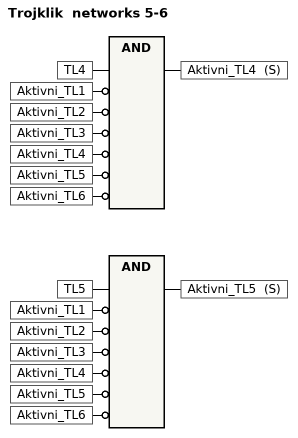
[picture p24: Trojklik (FBD) networks 5-6]
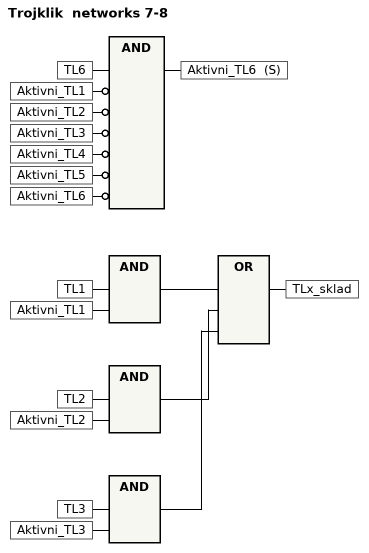
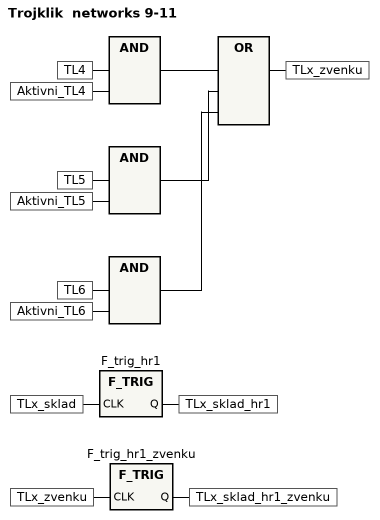
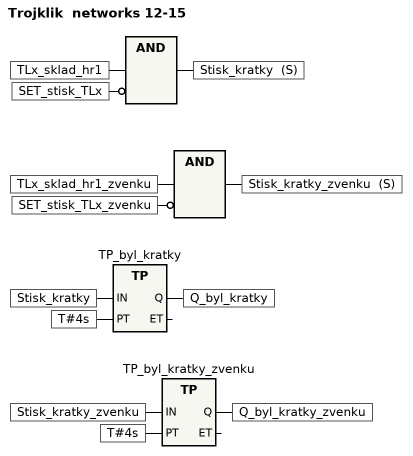
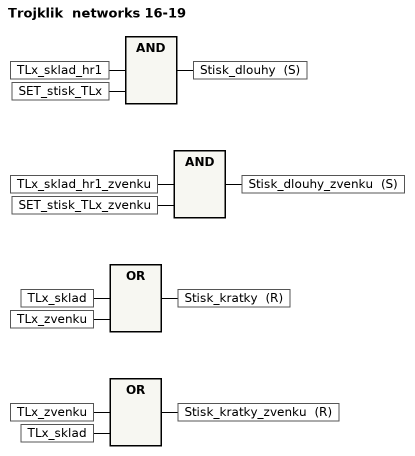
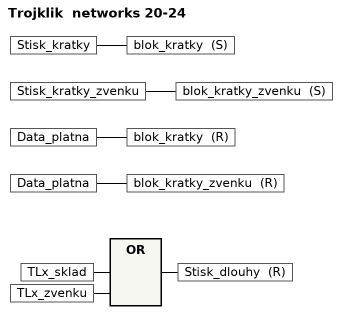
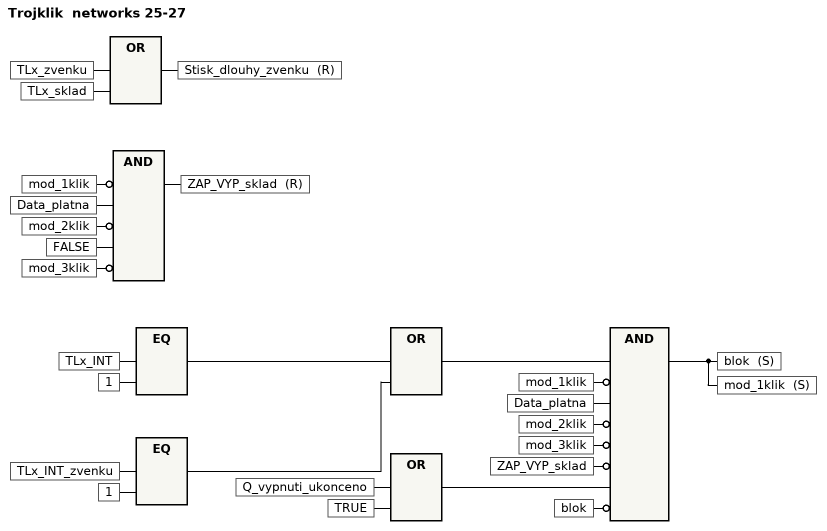
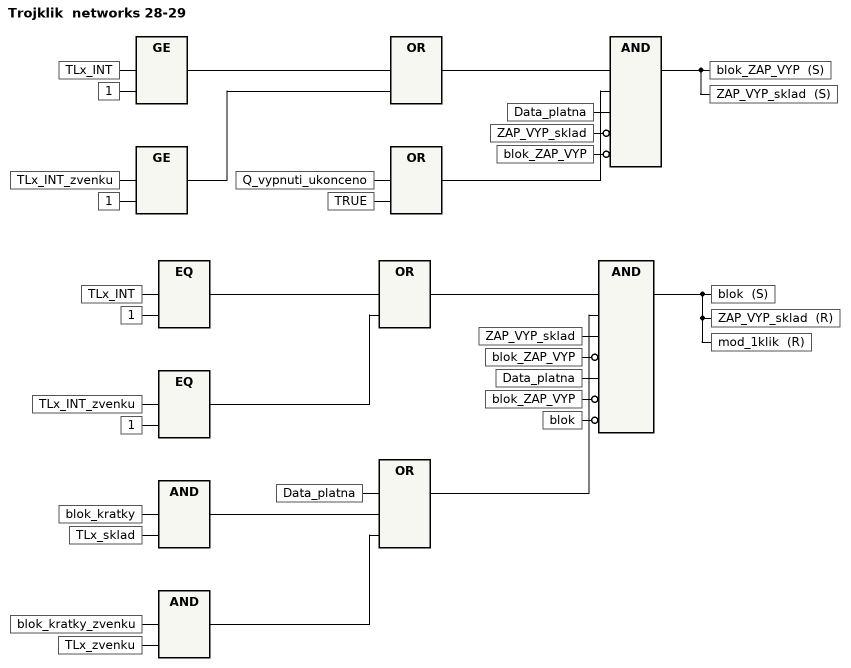
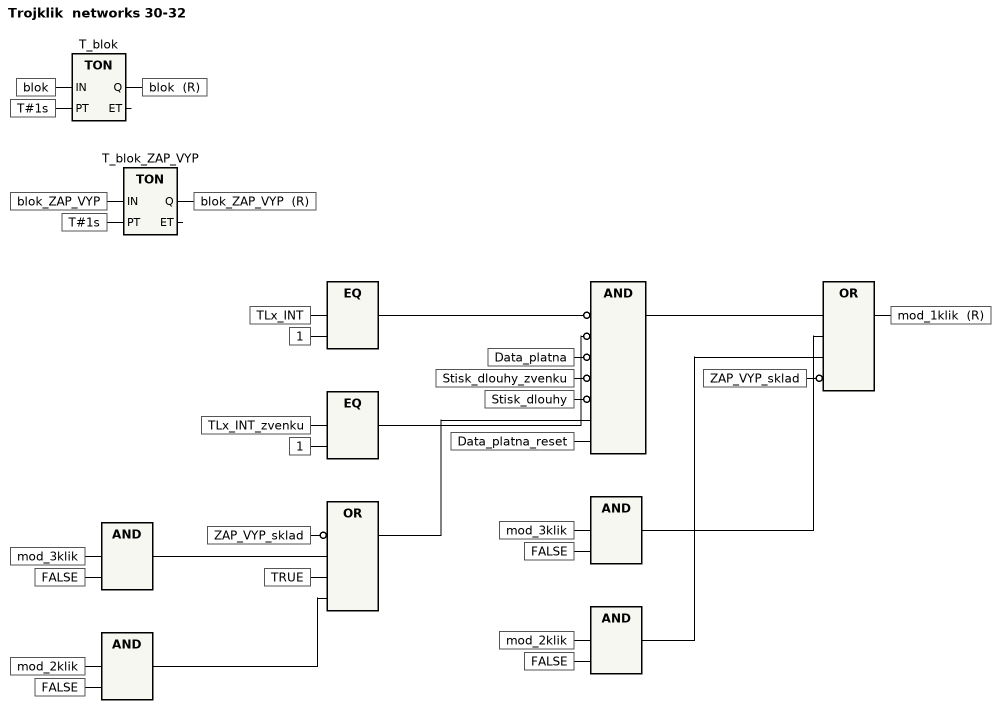
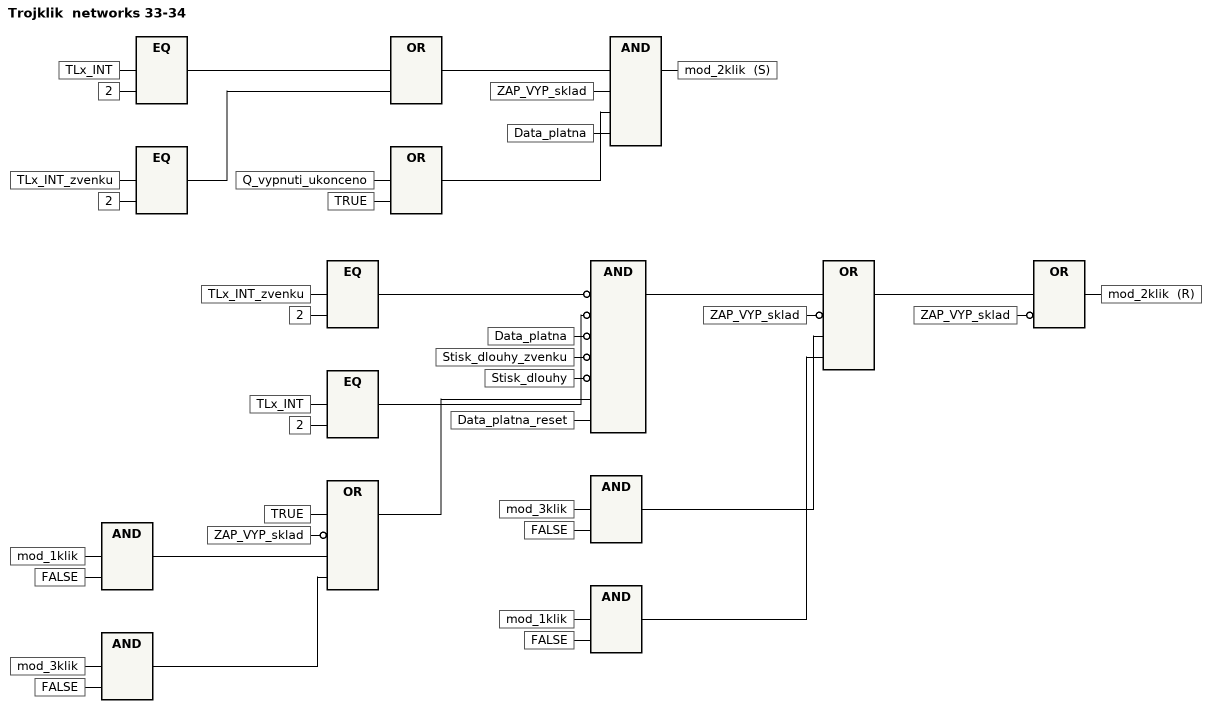
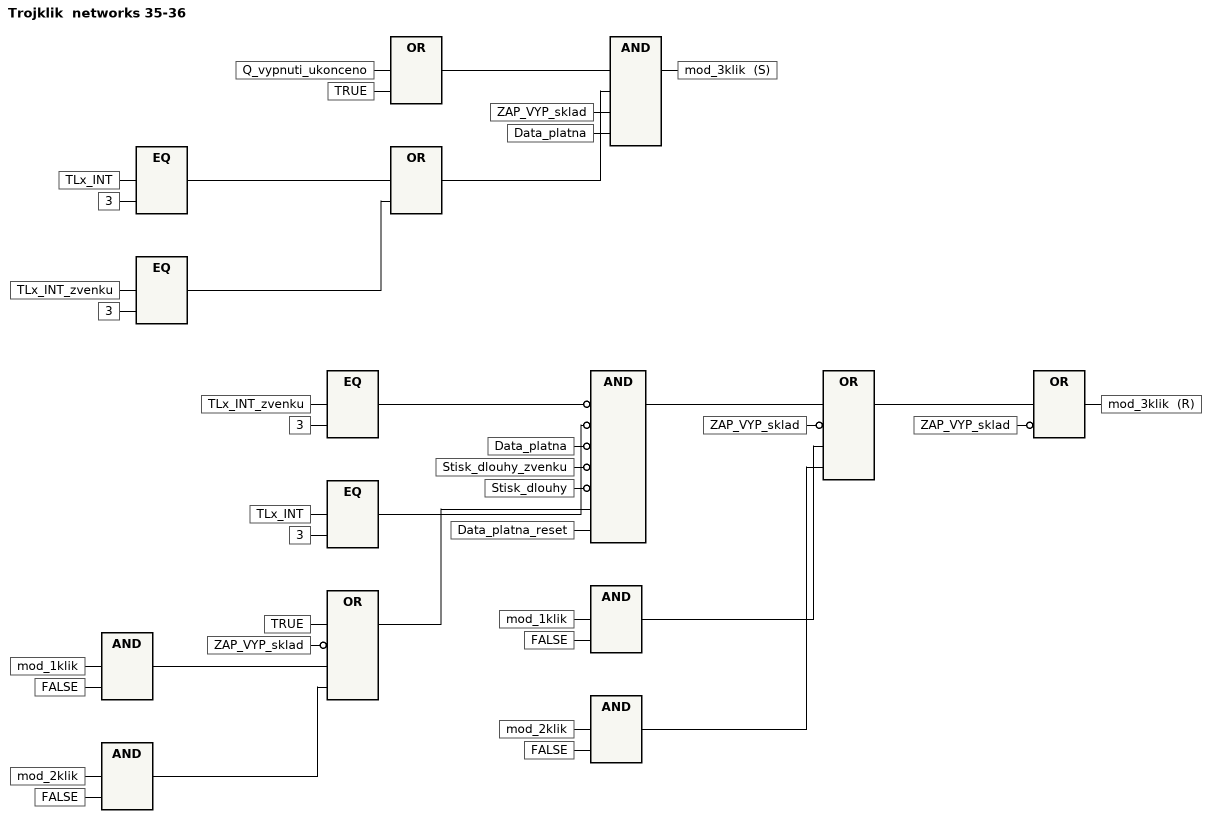
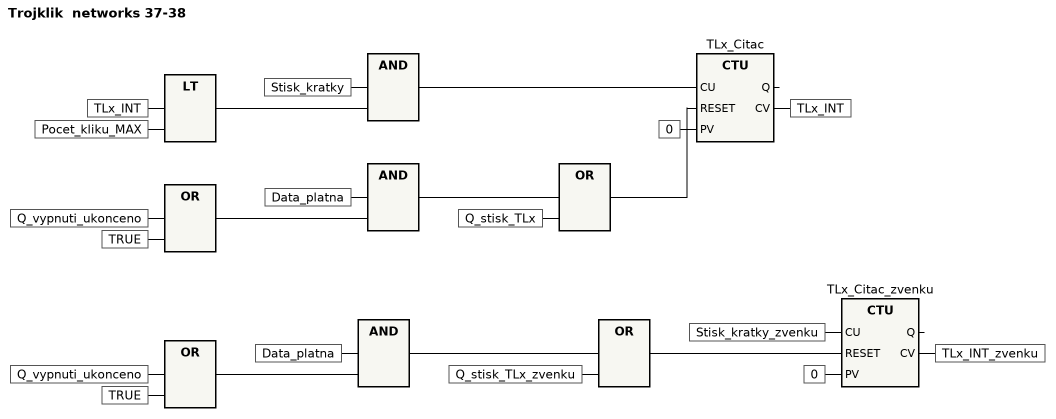
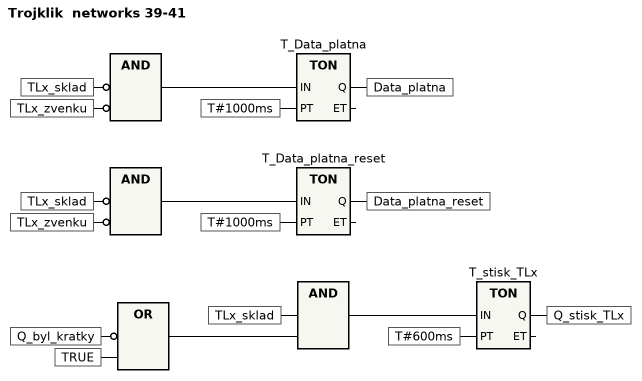
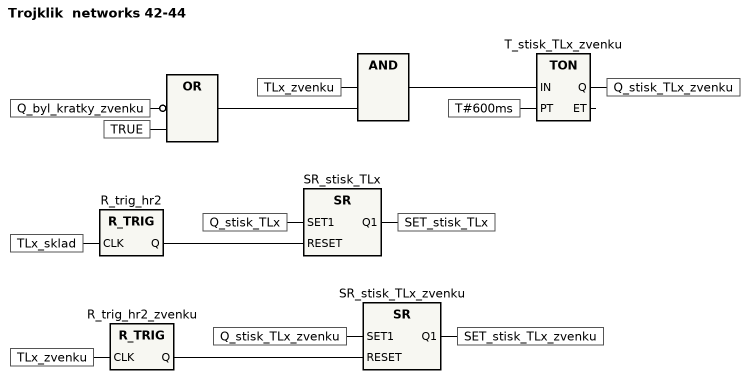
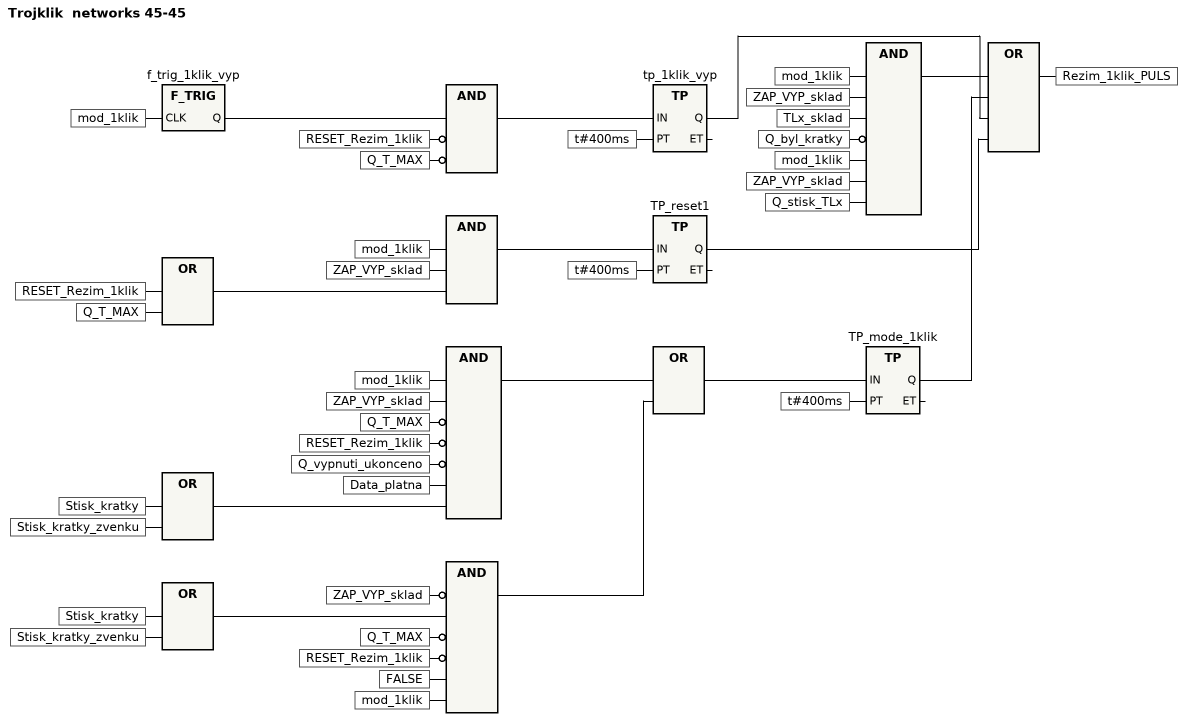
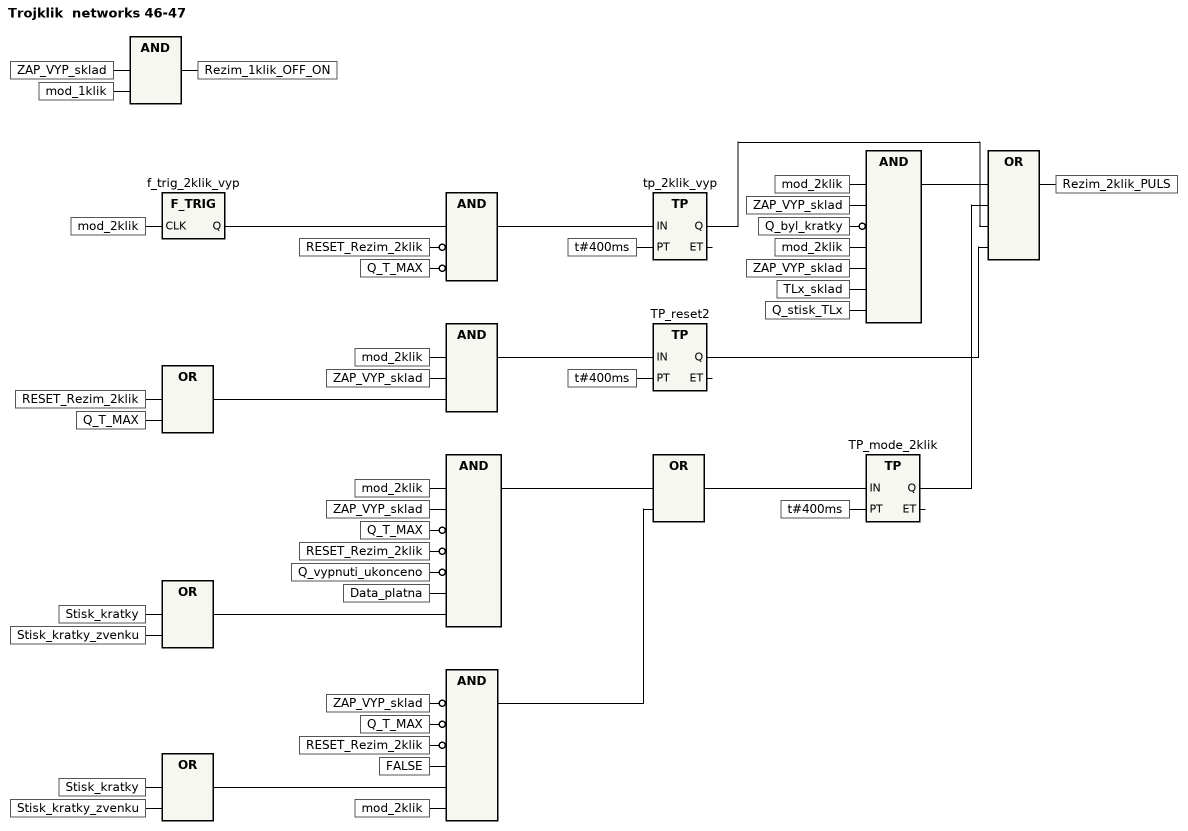
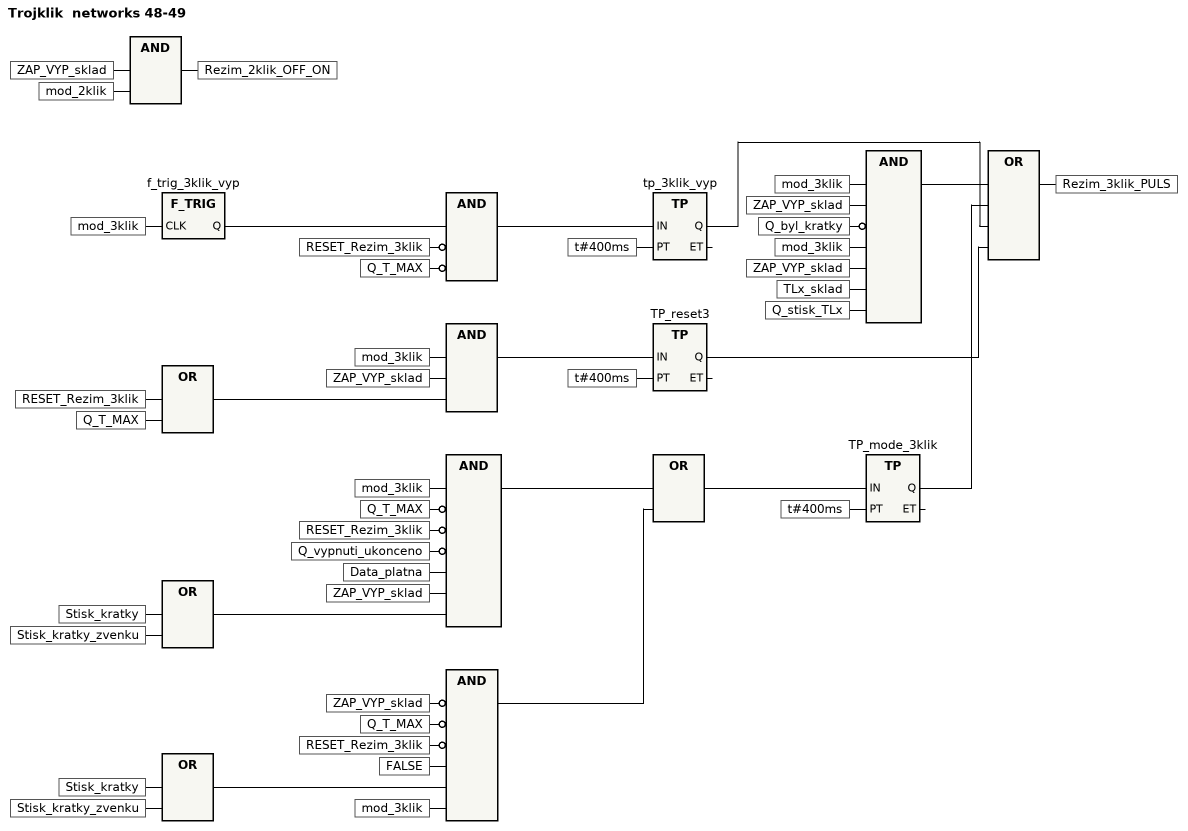
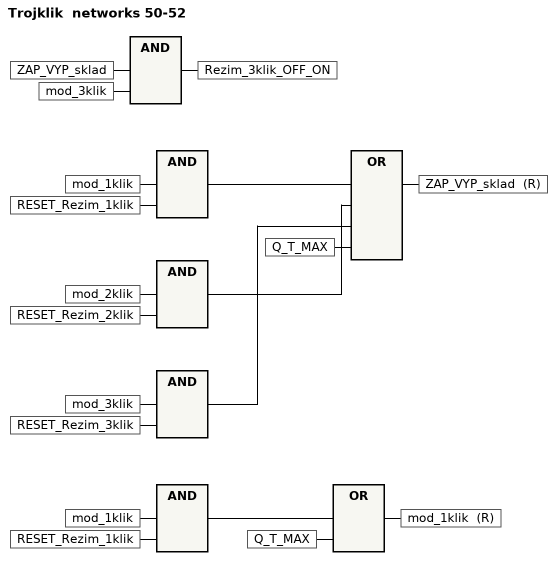
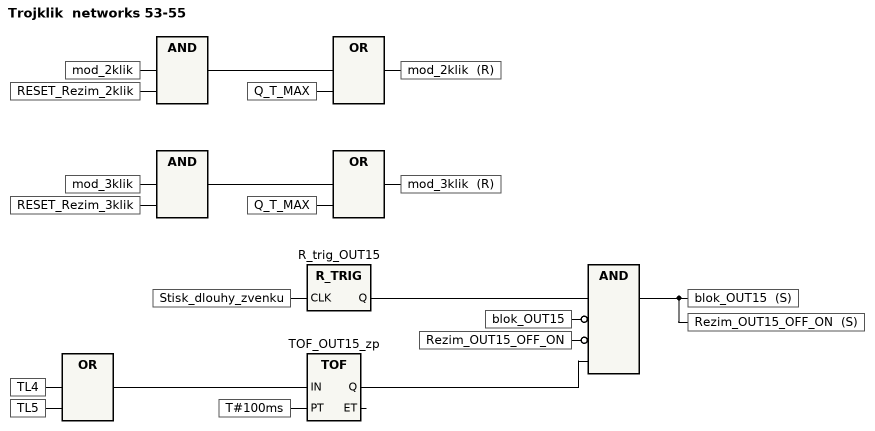
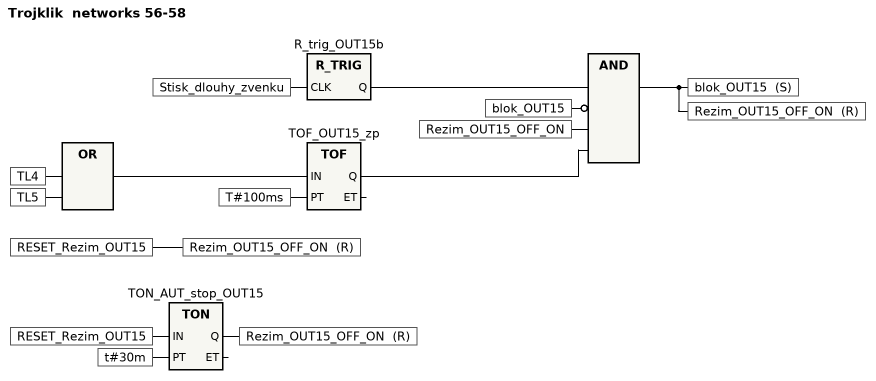
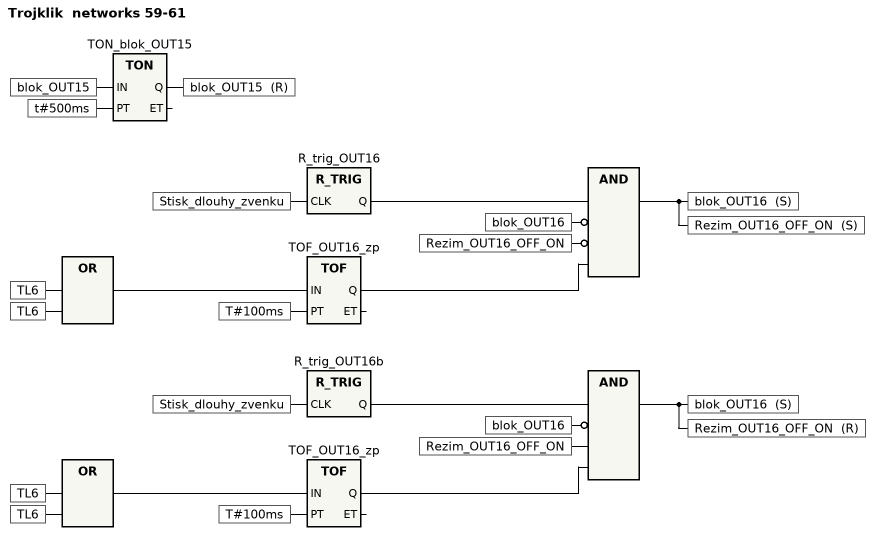
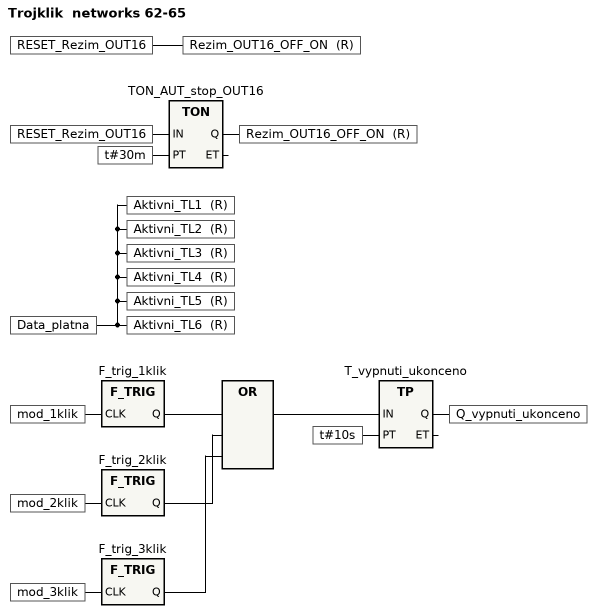
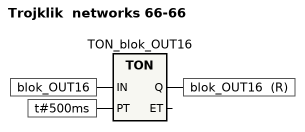
_FBD_ (* Function Block Diagram *)
NETWORK 1
	TP_T_max:TP(IN: T_max:TON(IN: AND(OR(Rezim_1klik_OFF_ON, Rezim_2klik_OFF_ON, Rezim_3klik_OFF_ON), AUT_vyp), PT: cas_vypnuti), PT: t#400ms) => Q_T_MAX
NETWORK 2
	AND(TL1, NOT Aktivni_TL1, NOT Aktivni_TL2, NOT Aktivni_TL3, NOT Aktivni_TL4, NOT Aktivni_TL5, NOT Aktivni_TL6) => S Aktivni_TL1
NETWORK 3
	AND(TL2, NOT Aktivni_TL1, NOT Aktivni_TL2, NOT Aktivni_TL3, NOT Aktivni_TL4, NOT Aktivni_TL5, NOT Aktivni_TL6) => S Aktivni_TL2
NETWORK 4
	AND(TL3, NOT Aktivni_TL1, NOT Aktivni_TL2, NOT Aktivni_TL3, NOT Aktivni_TL4, NOT Aktivni_TL5, NOT Aktivni_TL6) => S Aktivni_TL3
NETWORK 5
	AND(TL4, NOT Aktivni_TL1, NOT Aktivni_TL2, NOT Aktivni_TL3, NOT Aktivni_TL4, NOT Aktivni_TL5, NOT Aktivni_TL6) => S Aktivni_TL4
NETWORK 6
	AND(TL5, NOT Aktivni_TL1, NOT Aktivni_TL2, NOT Aktivni_TL3, NOT Aktivni_TL4, NOT Aktivni_TL5, NOT Aktivni_TL6) => S Aktivni_TL5
NETWORK 7
	AND(TL6, NOT Aktivni_TL1, NOT Aktivni_TL2, NOT Aktivni_TL3, NOT Aktivni_TL4, NOT Aktivni_TL5, NOT Aktivni_TL6) => S Aktivni_TL6
NETWORK 8
	OR(AND(TL1, Aktivni_TL1), AND(TL2, Aktivni_TL2), AND(TL3, Aktivni_TL3)) => TLx_sklad
NETWORK 9
	OR(AND(TL4, Aktivni_TL4), AND(TL5, Aktivni_TL5), AND(TL6, Aktivni_TL6)) => TLx_zvenku
NETWORK 10
	F_trig_hr1:F_TRIG(CLK: TLx_sklad) => TLx_sklad_hr1
NETWORK 11
	F_trig_hr1_zvenku:F_TRIG(CLK: TLx_zvenku) => TLx_sklad_hr1_zvenku
NETWORK 12
	AND(TLx_sklad_hr1, NOT SET_stisk_TLx) => S Stisk_kratky
NETWORK 13
	AND(TLx_sklad_hr1_zvenku, NOT SET_stisk_TLx_zvenku) => S Stisk_kratky_zvenku
NETWORK 14
	TP_byl_kratky:TP(IN: Stisk_kratky, PT: T#4s) => Q_byl_kratky
NETWORK 15
	TP_byl_kratky_zvenku:TP(IN: Stisk_kratky_zvenku, PT: T#4s) => Q_byl_kratky_zvenku
NETWORK 16
	AND(TLx_sklad_hr1, SET_stisk_TLx) => S Stisk_dlouhy
NETWORK 17
	AND(TLx_sklad_hr1_zvenku, SET_stisk_TLx_zvenku) => S Stisk_dlouhy_zvenku
NETWORK 18
	OR(TLx_sklad, TLx_zvenku) => R Stisk_kratky
NETWORK 19
	OR(TLx_zvenku, TLx_sklad) => R Stisk_kratky_zvenku
NETWORK 20
	Stisk_kratky => S blok_kratky
NETWORK 21
	Stisk_kratky_zvenku => S blok_kratky_zvenku
NETWORK 22
	Data_platna => R blok_kratky
NETWORK 23
	Data_platna => R blok_kratky_zvenku
NETWORK 24
	OR(TLx_sklad, TLx_zvenku) => R Stisk_dlouhy
NETWORK 25
	OR(TLx_zvenku, TLx_sklad) => R Stisk_dlouhy_zvenku
NETWORK 26
	AND(NOT mod_1klik, Data_platna, NOT mod_2klik, FALSE, NOT mod_3klik) => R ZAP_VYP_sklad
NETWORK 27
	AND(OR(EQ(TLx_INT, 1), EQ(TLx_INT_zvenku, 1)), NOT mod_1klik, Data_platna, NOT mod_2klik, NOT mod_3klik, NOT ZAP_VYP_sklad, OR(Q_vypnuti_ukonceno, TRUE), NOT blok) => S blok, S mod_1klik
NETWORK 28
	AND(OR(GE(TLx_INT, 1), GE(TLx_INT_zvenku, 1)), OR(Q_vypnuti_ukonceno, TRUE), Data_platna, NOT ZAP_VYP_sklad, NOT blok_ZAP_VYP) => S blok_ZAP_VYP, S ZAP_VYP_sklad
NETWORK 29
	AND(OR(EQ(TLx_INT, 1), EQ(TLx_INT_zvenku, 1)), OR(Data_platna, AND(blok_kratky, TLx_sklad), AND(blok_kratky_zvenku, TLx_zvenku)), ZAP_VYP_sklad, NOT blok_ZAP_VYP, Data_platna, NOT blok_ZAP_VYP, NOT blok) => S blok, R ZAP_VYP_sklad, R mod_1klik
NETWORK 30
	T_blok:TON(IN: blok, PT: T#1s) => R blok
NETWORK 31
	T_blok_ZAP_VYP:TON(IN: blok_ZAP_VYP, PT: T#1s) => R blok_ZAP_VYP
NETWORK 32
	OR(AND(NOT EQ(TLx_INT, 1), NOT EQ(TLx_INT_zvenku, 1), NOT Data_platna, NOT Stisk_dlouhy_zvenku, NOT Stisk_dlouhy, OR(NOT ZAP_VYP_sklad, AND(mod_3klik, FALSE), TRUE, AND(mod_2klik, FALSE)), Data_platna_reset), AND(mod_3klik, FALSE), AND(mod_2klik, FALSE), NOT ZAP_VYP_sklad) => R mod_1klik
NETWORK 33
	AND(OR(EQ(TLx_INT, 2), EQ(TLx_INT_zvenku, 2)), ZAP_VYP_sklad, OR(Q_vypnuti_ukonceno, TRUE), Data_platna) => S mod_2klik
NETWORK 34
	OR(OR(AND(NOT EQ(TLx_INT_zvenku, 2), NOT EQ(TLx_INT, 2), NOT Data_platna, NOT Stisk_dlouhy_zvenku, NOT Stisk_dlouhy, OR(TRUE, NOT ZAP_VYP_sklad, AND(mod_1klik, FALSE), AND(mod_3klik, FALSE)), Data_platna_reset), NOT ZAP_VYP_sklad, AND(mod_3klik, FALSE), AND(mod_1klik, FALSE)), NOT ZAP_VYP_sklad) => R mod_2klik
NETWORK 35
	AND(OR(Q_vypnuti_ukonceno, TRUE), OR(EQ(TLx_INT, 3), EQ(TLx_INT_zvenku, 3)), ZAP_VYP_sklad, Data_platna) => S mod_3klik
NETWORK 36
	OR(OR(AND(NOT EQ(TLx_INT_zvenku, 3), NOT EQ(TLx_INT, 3), NOT Data_platna, NOT Stisk_dlouhy_zvenku, NOT Stisk_dlouhy, OR(TRUE, NOT ZAP_VYP_sklad, AND(mod_1klik, FALSE), AND(mod_2klik, FALSE)), Data_platna_reset), NOT ZAP_VYP_sklad, AND(mod_1klik, FALSE), AND(mod_2klik, FALSE)), NOT ZAP_VYP_sklad) => R mod_3klik
NETWORK 37
	TLx_Citac:CTU(CU: AND(Stisk_kratky, LT(TLx_INT, Pocet_kliku_MAX)), RESET: OR(AND(Data_platna, OR(Q_vypnuti_ukonceno, TRUE)), Q_stisk_TLx), PV: 0, CV => TLx_INT)
NETWORK 38
	TLx_Citac_zvenku:CTU(CU: Stisk_kratky_zvenku, RESET: OR(AND(Data_platna, OR(Q_vypnuti_ukonceno, TRUE)), Q_stisk_TLx_zvenku), PV: 0, CV => TLx_INT_zvenku)
NETWORK 39 (* Data platna *)
	T_Data_platna:TON(IN: AND(NOT TLx_sklad, NOT TLx_zvenku), PT: T#1000ms) => Data_platna
NETWORK 40 (* Data platna *)
	T_Data_platna_reset:TON(IN: AND(NOT TLx_sklad, NOT TLx_zvenku), PT: T#1000ms) => Data_platna_reset
NETWORK 41 (* delka stisku TLx *)
	T_stisk_TLx:TON(IN: AND(TLx_sklad, OR(NOT Q_byl_kratky, TRUE)), PT: T#600ms) => Q_stisk_TLx
NETWORK 42 (* delka stisku TLx *)
	T_stisk_TLx_zvenku:TON(IN: AND(TLx_zvenku, OR(NOT Q_byl_kratky_zvenku, TRUE)), PT: T#600ms) => Q_stisk_TLx_zvenku
NETWORK 43
	SR_stisk_TLx:SR(SET1: Q_stisk_TLx, RESET: R_trig_hr2:R_TRIG(CLK: TLx_sklad)) => SET_stisk_TLx
NETWORK 44
	SR_stisk_TLx_zvenku:SR(SET1: Q_stisk_TLx_zvenku, RESET: R_trig_hr2_zvenku:R_TRIG(CLK: TLx_zvenku)) => SET_stisk_TLx_zvenku
NETWORK 45
	OR(AND(mod_1klik, ZAP_VYP_sklad, TLx_sklad, NOT Q_byl_kratky, mod_1klik, ZAP_VYP_sklad, Q_stisk_TLx), TP_mode_1klik:TP(IN: OR(AND(mod_1klik, ZAP_VYP_sklad, NOT Q_T_MAX, NOT RESET_Rezim_1klik, NOT Q_vypnuti_ukonceno, Data_platna, OR(Stisk_kratky, Stisk_kratky_zvenku)), AND(NOT ZAP_VYP_sklad, OR(Stisk_kratky, Stisk_kratky_zvenku), NOT Q_T_MAX, NOT RESET_Rezim_1klik, FALSE, mod_1klik)), PT: t#400ms), tp_1klik_vyp:TP(IN: AND(f_trig_1klik_vyp:F_TRIG(CLK: mod_1klik), NOT RESET_Rezim_1klik, NOT Q_T_MAX), PT: t#400ms), TP_reset1:TP(IN: AND(mod_1klik, ZAP_VYP_sklad, OR(RESET_Rezim_1klik, Q_T_MAX)), PT: t#400ms)) => Rezim_1klik_PULS
NETWORK 46
	AND(ZAP_VYP_sklad, mod_1klik) => Rezim_1klik_OFF_ON
NETWORK 47
	OR(AND(mod_2klik, ZAP_VYP_sklad, NOT Q_byl_kratky, mod_2klik, ZAP_VYP_sklad, TLx_sklad, Q_stisk_TLx), TP_mode_2klik:TP(IN: OR(AND(mod_2klik, ZAP_VYP_sklad, NOT Q_T_MAX, NOT RESET_Rezim_2klik, NOT Q_vypnuti_ukonceno, Data_platna, OR(Stisk_kratky, Stisk_kratky_zvenku)), AND(NOT ZAP_VYP_sklad, NOT Q_T_MAX, NOT RESET_Rezim_2klik, FALSE, OR(Stisk_kratky, Stisk_kratky_zvenku), mod_2klik)), PT: t#400ms), tp_2klik_vyp:TP(IN: AND(f_trig_2klik_vyp:F_TRIG(CLK: mod_2klik), NOT RESET_Rezim_2klik, NOT Q_T_MAX), PT: t#400ms), TP_reset2:TP(IN: AND(mod_2klik, ZAP_VYP_sklad, OR(RESET_Rezim_2klik, Q_T_MAX)), PT: t#400ms)) => Rezim_2klik_PULS
NETWORK 48
	AND(ZAP_VYP_sklad, mod_2klik) => Rezim_2klik_OFF_ON
NETWORK 49
	OR(AND(mod_3klik, ZAP_VYP_sklad, NOT Q_byl_kratky, mod_3klik, ZAP_VYP_sklad, TLx_sklad, Q_stisk_TLx), TP_mode_3klik:TP(IN: OR(AND(mod_3klik, NOT Q_T_MAX, NOT RESET_Rezim_3klik, NOT Q_vypnuti_ukonceno, Data_platna, ZAP_VYP_sklad, OR(Stisk_kratky, Stisk_kratky_zvenku)), AND(NOT ZAP_VYP_sklad, NOT Q_T_MAX, NOT RESET_Rezim_3klik, FALSE, OR(Stisk_kratky, Stisk_kratky_zvenku), mod_3klik)), PT: t#400ms), tp_3klik_vyp:TP(IN: AND(f_trig_3klik_vyp:F_TRIG(CLK: mod_3klik), NOT RESET_Rezim_3klik, NOT Q_T_MAX), PT: t#400ms), TP_reset3:TP(IN: AND(mod_3klik, ZAP_VYP_sklad, OR(RESET_Rezim_3klik, Q_T_MAX)), PT: t#400ms)) => Rezim_3klik_PULS
NETWORK 50
	AND(ZAP_VYP_sklad, mod_3klik) => Rezim_3klik_OFF_ON
NETWORK 51
	OR(AND(mod_1klik, RESET_Rezim_1klik), AND(mod_2klik, RESET_Rezim_2klik), AND(mod_3klik, RESET_Rezim_3klik), Q_T_MAX) => R ZAP_VYP_sklad
NETWORK 52
	OR(AND(mod_1klik, RESET_Rezim_1klik), Q_T_MAX) => R mod_1klik
NETWORK 53
	OR(AND(mod_2klik, RESET_Rezim_2klik), Q_T_MAX) => R mod_2klik
NETWORK 54
	OR(AND(mod_3klik, RESET_Rezim_3klik), Q_T_MAX) => R mod_3klik
NETWORK 55
	AND(R_trig_OUT15:R_TRIG(CLK: Stisk_dlouhy_zvenku), NOT blok_OUT15, NOT Rezim_OUT15_OFF_ON, TOF_OUT15_zp:TOF(IN: OR(TL4, TL5), PT: T#100ms)) => S blok_OUT15, S Rezim_OUT15_OFF_ON
NETWORK 56
	AND(R_trig_OUT15b:R_TRIG(CLK: Stisk_dlouhy_zvenku), NOT blok_OUT15, Rezim_OUT15_OFF_ON, TOF_OUT15_zp:TOF(IN: OR(TL4, TL5), PT: T#100ms)) => S blok_OUT15, R Rezim_OUT15_OFF_ON
NETWORK 57
	RESET_Rezim_OUT15 => R Rezim_OUT15_OFF_ON
NETWORK 58
	TON_AUT_stop_OUT15:TON(IN: RESET_Rezim_OUT15, PT: t#30m) => R Rezim_OUT15_OFF_ON
NETWORK 59
	TON_blok_OUT15:TON(IN: blok_OUT15, PT: t#500ms) => R blok_OUT15
NETWORK 60
	AND(R_trig_OUT16:R_TRIG(CLK: Stisk_dlouhy_zvenku), NOT blok_OUT16, NOT Rezim_OUT16_OFF_ON, TOF_OUT16_zp:TOF(IN: OR(TL6, TL6), PT: T#100ms)) => S blok_OUT16, S Rezim_OUT16_OFF_ON
NETWORK 61
	AND(R_trig_OUT16b:R_TRIG(CLK: Stisk_dlouhy_zvenku), NOT blok_OUT16, Rezim_OUT16_OFF_ON, TOF_OUT16_zp:TOF(IN: OR(TL6, TL6), PT: T#100ms)) => S blok_OUT16, R Rezim_OUT16_OFF_ON
NETWORK 62
	RESET_Rezim_OUT16 => R Rezim_OUT16_OFF_ON
NETWORK 63
	TON_AUT_stop_OUT16:TON(IN: RESET_Rezim_OUT16, PT: t#30m) => R Rezim_OUT16_OFF_ON
NETWORK 64
	Data_platna => R Aktivni_TL1, R Aktivni_TL2, R Aktivni_TL3, R Aktivni_TL4, R Aktivni_TL5, R Aktivni_TL6
NETWORK 65
	T_vypnuti_ukonceno:TP(IN: OR(F_trig_1klik:F_TRIG(CLK: mod_1klik), F_trig_2klik:F_TRIG(CLK: mod_2klik), F_trig_3klik:F_TRIG(CLK: mod_3klik)), PT: t#10s) => Q_vypnuti_ukonceno
NETWORK 66
	TON_blok_OUT16:TON(IN: blok_OUT16, PT: t#500ms) => R blok_OUT16
_END_FBD_
(* the same logic as Structured Text *)
(* Network 1 *)
T_max(IN := (Rezim_1klik_OFF_ON OR Rezim_2klik_OFF_ON OR Rezim_3klik_OFF_ON) AND AUT_vyp, PT := cas_vypnuti);
TP_T_max(IN := T_max.Q, PT := t#400ms);
Q_T_MAX := TP_T_max.Q;
(* Network 2 *)
IF TL1 AND NOT Aktivni_TL1 AND NOT Aktivni_TL2 AND NOT Aktivni_TL3 AND NOT Aktivni_TL4 AND NOT Aktivni_TL5 AND NOT Aktivni_TL6 THEN Aktivni_TL1 := TRUE; END_IF;
(* Network 3 *)
IF TL2 AND NOT Aktivni_TL1 AND NOT Aktivni_TL2 AND NOT Aktivni_TL3 AND NOT Aktivni_TL4 AND NOT Aktivni_TL5 AND NOT Aktivni_TL6 THEN Aktivni_TL2 := TRUE; END_IF;
(* Network 4 *)
IF TL3 AND NOT Aktivni_TL1 AND NOT Aktivni_TL2 AND NOT Aktivni_TL3 AND NOT Aktivni_TL4 AND NOT Aktivni_TL5 AND NOT Aktivni_TL6 THEN Aktivni_TL3 := TRUE; END_IF;
(* Network 5 *)
IF TL4 AND NOT Aktivni_TL1 AND NOT Aktivni_TL2 AND NOT Aktivni_TL3 AND NOT Aktivni_TL4 AND NOT Aktivni_TL5 AND NOT Aktivni_TL6 THEN Aktivni_TL4 := TRUE; END_IF;
(* Network 6 *)
IF TL5 AND NOT Aktivni_TL1 AND NOT Aktivni_TL2 AND NOT Aktivni_TL3 AND NOT Aktivni_TL4 AND NOT Aktivni_TL5 AND NOT Aktivni_TL6 THEN Aktivni_TL5 := TRUE; END_IF;
(* Network 7 *)
IF TL6 AND NOT Aktivni_TL1 AND NOT Aktivni_TL2 AND NOT Aktivni_TL3 AND NOT Aktivni_TL4 AND NOT Aktivni_TL5 AND NOT Aktivni_TL6 THEN Aktivni_TL6 := TRUE; END_IF;
(* Network 8 *)
TLx_sklad := (TL1 AND Aktivni_TL1) OR (TL2 AND Aktivni_TL2) OR (TL3 AND Aktivni_TL3);
(* Network 9 *)
TLx_zvenku := (TL4 AND Aktivni_TL4) OR (TL5 AND Aktivni_TL5) OR (TL6 AND Aktivni_TL6);
(* Network 10 *)
F_trig_hr1(CLK := TLx_sklad);
TLx_sklad_hr1 := F_trig_hr1.Q;
(* Network 11 *)
F_trig_hr1_zvenku(CLK := TLx_zvenku);
TLx_sklad_hr1_zvenku := F_trig_hr1_zvenku.Q;
(* Network 12 *)
IF TLx_sklad_hr1 AND NOT SET_stisk_TLx THEN Stisk_kratky := TRUE; END_IF;
(* Network 13 *)
IF TLx_sklad_hr1_zvenku AND NOT SET_stisk_TLx_zvenku THEN Stisk_kratky_zvenku := TRUE; END_IF;
(* Network 14 *)
TP_byl_kratky(IN := Stisk_kratky, PT := T#4s);
Q_byl_kratky := TP_byl_kratky.Q;
(* Network 15 *)
TP_byl_kratky_zvenku(IN := Stisk_kratky_zvenku, PT := T#4s);
Q_byl_kratky_zvenku := TP_byl_kratky_zvenku.Q;
(* Network 16 *)
IF TLx_sklad_hr1 AND SET_stisk_TLx THEN Stisk_dlouhy := TRUE; END_IF;
(* Network 17 *)
IF TLx_sklad_hr1_zvenku AND SET_stisk_TLx_zvenku THEN Stisk_dlouhy_zvenku := TRUE; END_IF;
(* Network 18 *)
IF TLx_sklad OR TLx_zvenku THEN Stisk_kratky := FALSE; END_IF;
(* Network 19 *)
IF TLx_zvenku OR TLx_sklad THEN Stisk_kratky_zvenku := FALSE; END_IF;
(* Network 20 *)
IF Stisk_kratky THEN blok_kratky := TRUE; END_IF;
(* Network 21 *)
IF Stisk_kratky_zvenku THEN blok_kratky_zvenku := TRUE; END_IF;
(* Network 22 *)
IF Data_platna THEN blok_kratky := FALSE; END_IF;
(* Network 23 *)
IF Data_platna THEN blok_kratky_zvenku := FALSE; END_IF;
(* Network 24 *)
IF TLx_sklad OR TLx_zvenku THEN Stisk_dlouhy := FALSE; END_IF;
(* Network 25 *)
IF TLx_zvenku OR TLx_sklad THEN Stisk_dlouhy_zvenku := FALSE; END_IF;
(* Network 26 *)
IF NOT mod_1klik AND Data_platna AND NOT mod_2klik AND FALSE AND NOT mod_3klik THEN ZAP_VYP_sklad := FALSE; END_IF;
(* Network 27 *)
_p1 := ((TLx_INT = 1) OR (TLx_INT_zvenku = 1)) AND NOT mod_1klik AND Data_platna AND NOT mod_2klik AND NOT mod_3klik AND NOT ZAP_VYP_sklad AND (Q_vypnuti_ukonceno OR TRUE) AND NOT blok;
IF _p1 THEN blok := TRUE; mod_1klik := TRUE; END_IF;
(* Network 28 *)
_p2 := ((TLx_INT >= 1) OR (TLx_INT_zvenku >= 1)) AND (Q_vypnuti_ukonceno OR TRUE) AND Data_platna AND NOT ZAP_VYP_sklad AND NOT blok_ZAP_VYP;
IF _p2 THEN blok_ZAP_VYP := TRUE; ZAP_VYP_sklad := TRUE; END_IF;
(* Network 29 *)
_p3 := ((TLx_INT = 1) OR (TLx_INT_zvenku = 1)) AND (Data_platna OR (blok_kratky AND TLx_sklad) OR (blok_kratky_zvenku AND TLx_zvenku)) AND ZAP_VYP_sklad AND NOT blok_ZAP_VYP AND Data_platna AND NOT blok_ZAP_VYP AND NOT blok;
IF _p3 THEN blok := TRUE; ZAP_VYP_sklad := FALSE; mod_1klik := FALSE; END_IF;
(* Network 30 *)
T_blok(IN := blok, PT := T#1s);
IF T_blok.Q THEN blok := FALSE; END_IF;
(* Network 31 *)
T_blok_ZAP_VYP(IN := blok_ZAP_VYP, PT := T#1s);
IF T_blok_ZAP_VYP.Q THEN blok_ZAP_VYP := FALSE; END_IF;
(* Network 32 *)
IF (NOT (TLx_INT = 1) AND NOT (TLx_INT_zvenku = 1) AND NOT Data_platna AND NOT Stisk_dlouhy_zvenku AND NOT Stisk_dlouhy AND (NOT ZAP_VYP_sklad OR (mod_3klik AND FALSE) OR TRUE OR (mod_2klik AND FALSE)) AND Data_platna_reset) OR (mod_3klik AND FALSE) OR (mod_2klik AND FALSE) OR NOT ZAP_VYP_sklad THEN mod_1klik := FALSE; END_IF;
(* Network 33 *)
IF ((TLx_INT = 2) OR (TLx_INT_zvenku = 2)) AND ZAP_VYP_sklad AND (Q_vypnuti_ukonceno OR TRUE) AND Data_platna THEN mod_2klik := TRUE; END_IF;
(* Network 34 *)
IF ((NOT (TLx_INT_zvenku = 2) AND NOT (TLx_INT = 2) AND NOT Data_platna AND NOT Stisk_dlouhy_zvenku AND NOT Stisk_dlouhy AND (TRUE OR NOT ZAP_VYP_sklad OR (mod_1klik AND FALSE) OR (mod_3klik AND FALSE)) AND Data_platna_reset) OR NOT ZAP_VYP_sklad OR (mod_3klik AND FALSE) OR (mod_1klik AND FALSE)) OR NOT ZAP_VYP_sklad THEN mod_2klik := FALSE; END_IF;
(* Network 35 *)
IF (Q_vypnuti_ukonceno OR TRUE) AND ((TLx_INT = 3) OR (TLx_INT_zvenku = 3)) AND ZAP_VYP_sklad AND Data_platna THEN mod_3klik := TRUE; END_IF;
(* Network 36 *)
IF ((NOT (TLx_INT_zvenku = 3) AND NOT (TLx_INT = 3) AND NOT Data_platna AND NOT Stisk_dlouhy_zvenku AND NOT Stisk_dlouhy AND (TRUE OR NOT ZAP_VYP_sklad OR (mod_1klik AND FALSE) OR (mod_2klik AND FALSE)) AND Data_platna_reset) OR NOT ZAP_VYP_sklad OR (mod_1klik AND FALSE) OR (mod_2klik AND FALSE)) OR NOT ZAP_VYP_sklad THEN mod_3klik := FALSE; END_IF;
(* Network 37 *)
TLx_Citac(CU := Stisk_kratky AND (TLx_INT < Pocet_kliku_MAX), RESET := (Data_platna AND (Q_vypnuti_ukonceno OR TRUE)) OR Q_stisk_TLx, PV := 0);
TLx_INT := TLx_Citac.CV;
(* Network 38 *)
TLx_Citac_zvenku(CU := Stisk_kratky_zvenku, RESET := (Data_platna AND (Q_vypnuti_ukonceno OR TRUE)) OR Q_stisk_TLx_zvenku, PV := 0);
TLx_INT_zvenku := TLx_Citac_zvenku.CV;
(* Network 39 *)
T_Data_platna(IN := NOT TLx_sklad AND NOT TLx_zvenku, PT := T#1000ms);
Data_platna := T_Data_platna.Q;
(* Network 40 *)
T_Data_platna_reset(IN := NOT TLx_sklad AND NOT TLx_zvenku, PT := T#1000ms);
Data_platna_reset := T_Data_platna_reset.Q;
(* Network 41: see the listing above *)
(* Network 42: see the listing above *)
(* Network 43 *)
R_trig_hr2(CLK := TLx_sklad);
SR_stisk_TLx(SET1 := Q_stisk_TLx, RESET := R_trig_hr2.Q);
SET_stisk_TLx := SR_stisk_TLx.Q1;
(* Network 44 *)
R_trig_hr2_zvenku(CLK := TLx_zvenku);
SR_stisk_TLx_zvenku(SET1 := Q_stisk_TLx_zvenku, RESET := R_trig_hr2_zvenku.Q);
SET_stisk_TLx_zvenku := SR_stisk_TLx_zvenku.Q1;
(* Network 45 *)
TP_mode_1klik(IN := (mod_1klik AND ZAP_VYP_sklad AND NOT Q_T_MAX AND NOT RESET_Rezim_1klik AND NOT Q_vypnuti_ukonceno AND Data_platna AND (Stisk_kratky OR Stisk_kratky_zvenku)) OR (NOT ZAP_VYP_sklad AND (Stisk_kratky OR Stisk_kratky_zvenku) AND NOT Q_T_MAX AND NOT RESET_Rezim_1klik AND FALSE AND mod_1klik), PT := t#400ms);
f_trig_1klik_vyp(CLK := mod_1klik);
tp_1klik_vyp(IN := f_trig_1klik_vyp.Q AND NOT RESET_Rezim_1klik AND NOT Q_T_MAX, PT := t#400ms);
TP_reset1(IN := mod_1klik AND ZAP_VYP_sklad AND (RESET_Rezim_1klik OR Q_T_MAX), PT := t#400ms);
Rezim_1klik_PULS := (mod_1klik AND ZAP_VYP_sklad AND TLx_sklad AND NOT Q_byl_kratky AND mod_1klik AND ZAP_VYP_sklad AND Q_stisk_TLx) OR TP_mode_1klik.Q OR tp_1klik_vyp.Q OR TP_reset1.Q;
(* Network 46 *)
Rezim_1klik_OFF_ON := ZAP_VYP_sklad AND mod_1klik;
(* Network 47 *)
TP_mode_2klik(IN := (mod_2klik AND ZAP_VYP_sklad AND NOT Q_T_MAX AND NOT RESET_Rezim_2klik AND NOT Q_vypnuti_ukonceno AND Data_platna AND (Stisk_kratky OR Stisk_kratky_zvenku)) OR (NOT ZAP_VYP_sklad AND NOT Q_T_MAX AND NOT RESET_Rezim_2klik AND FALSE AND (Stisk_kratky OR Stisk_kratky_zvenku) AND mod_2klik), PT := t#400ms);
f_trig_2klik_vyp(CLK := mod_2klik);
tp_2klik_vyp(IN := f_trig_2klik_vyp.Q AND NOT RESET_Rezim_2klik AND NOT Q_T_MAX, PT := t#400ms);
TP_reset2(IN := mod_2klik AND ZAP_VYP_sklad AND (RESET_Rezim_2klik OR Q_T_MAX), PT := t#400ms);
Rezim_2klik_PULS := (mod_2klik AND ZAP_VYP_sklad AND NOT Q_byl_kratky AND mod_2klik AND ZAP_VYP_sklad AND TLx_sklad AND Q_stisk_TLx) OR TP_mode_2klik.Q OR tp_2klik_vyp.Q OR TP_reset2.Q;
(* Network 48 *)
Rezim_2klik_OFF_ON := ZAP_VYP_sklad AND mod_2klik;
(* Network 49 *)
TP_mode_3klik(IN := (mod_3klik AND NOT Q_T_MAX AND NOT RESET_Rezim_3klik AND NOT Q_vypnuti_ukonceno AND Data_platna AND ZAP_VYP_sklad AND (Stisk_kratky OR Stisk_kratky_zvenku)) OR (NOT ZAP_VYP_sklad AND NOT Q_T_MAX AND NOT RESET_Rezim_3klik AND FALSE AND (Stisk_kratky OR Stisk_kratky_zvenku) AND mod_3klik), PT := t#400ms);
f_trig_3klik_vyp(CLK := mod_3klik);
tp_3klik_vyp(IN := f_trig_3klik_vyp.Q AND NOT RESET_Rezim_3klik AND NOT Q_T_MAX, PT := t#400ms);
TP_reset3(IN := mod_3klik AND ZAP_VYP_sklad AND (RESET_Rezim_3klik OR Q_T_MAX), PT := t#400ms);
Rezim_3klik_PULS := (mod_3klik AND ZAP_VYP_sklad AND NOT Q_byl_kratky AND mod_3klik AND ZAP_VYP_sklad AND TLx_sklad AND Q_stisk_TLx) OR TP_mode_3klik.Q OR tp_3klik_vyp.Q OR TP_reset3.Q;
(* Network 50 *)
Rezim_3klik_OFF_ON := ZAP_VYP_sklad AND mod_3klik;
(* Network 51 *)
IF (mod_1klik AND RESET_Rezim_1klik) OR (mod_2klik AND RESET_Rezim_2klik) OR (mod_3klik AND RESET_Rezim_3klik) OR Q_T_MAX THEN ZAP_VYP_sklad := FALSE; END_IF;
(* Network 52 *)
IF (mod_1klik AND RESET_Rezim_1klik) OR Q_T_MAX THEN mod_1klik := FALSE; END_IF;
(* Network 53 *)
IF (mod_2klik AND RESET_Rezim_2klik) OR Q_T_MAX THEN mod_2klik := FALSE; END_IF;
(* Network 54 *)
IF (mod_3klik AND RESET_Rezim_3klik) OR Q_T_MAX THEN mod_3klik := FALSE; END_IF;
(* Network 55 *)
R_trig_OUT15(CLK := Stisk_dlouhy_zvenku);
TOF_OUT15_zp(IN := TL4 OR TL5, PT := T#100ms);
_p4 := R_trig_OUT15.Q AND NOT blok_OUT15 AND NOT Rezim_OUT15_OFF_ON AND TOF_OUT15_zp.Q;
IF _p4 THEN blok_OUT15 := TRUE; Rezim_OUT15_OFF_ON := TRUE; END_IF;
(* Network 56 *)
R_trig_OUT15b(CLK := Stisk_dlouhy_zvenku);
TOF_OUT15_zp(IN := TL4 OR TL5, PT := T#100ms);
_p5 := R_trig_OUT15b.Q AND NOT blok_OUT15 AND Rezim_OUT15_OFF_ON AND TOF_OUT15_zp.Q;
IF _p5 THEN blok_OUT15 := TRUE; Rezim_OUT15_OFF_ON := FALSE; END_IF;
(* Network 57 *)
IF RESET_Rezim_OUT15 THEN Rezim_OUT15_OFF_ON := FALSE; END_IF;
(* Network 58 *)
TON_AUT_stop_OUT15(IN := RESET_Rezim_OUT15, PT := t#30m);
IF TON_AUT_stop_OUT15.Q THEN Rezim_OUT15_OFF_ON := FALSE; END_IF;
(* Network 59 *)
TON_blok_OUT15(IN := blok_OUT15, PT := t#500ms);
IF TON_blok_OUT15.Q THEN blok_OUT15 := FALSE; END_IF;
(* Network 60 *)
R_trig_OUT16(CLK := Stisk_dlouhy_zvenku);
TOF_OUT16_zp(IN := TL6 OR TL6, PT := T#100ms);
_p6 := R_trig_OUT16.Q AND NOT blok_OUT16 AND NOT Rezim_OUT16_OFF_ON AND TOF_OUT16_zp.Q;
IF _p6 THEN blok_OUT16 := TRUE; Rezim_OUT16_OFF_ON := TRUE; END_IF;
(* Network 61 *)
R_trig_OUT16b(CLK := Stisk_dlouhy_zvenku);
TOF_OUT16_zp(IN := TL6 OR TL6, PT := T#100ms);
_p7 := R_trig_OUT16b.Q AND NOT blok_OUT16 AND Rezim_OUT16_OFF_ON AND TOF_OUT16_zp.Q;
IF _p7 THEN blok_OUT16 := TRUE; Rezim_OUT16_OFF_ON := FALSE; END_IF;
(* Network 62 *)
IF RESET_Rezim_OUT16 THEN Rezim_OUT16_OFF_ON := FALSE; END_IF;
(* Network 63 *)
TON_AUT_stop_OUT16(IN := RESET_Rezim_OUT16, PT := t#30m);
IF TON_AUT_stop_OUT16.Q THEN Rezim_OUT16_OFF_ON := FALSE; END_IF;
(* Network 64 *)
IF Data_platna THEN Aktivni_TL1 := FALSE; Aktivni_TL2 := FALSE; Aktivni_TL3 := FALSE; Aktivni_TL4 := FALSE; Aktivni_TL5 := FALSE; Aktivni_TL6 := FALSE; END_IF;
(* Network 65 *)
F_trig_1klik(CLK := mod_1klik);
F_trig_2klik(CLK := mod_2klik);
F_trig_3klik(CLK := mod_3klik);
T_vypnuti_ukonceno(IN := F_trig_1klik.Q OR F_trig_2klik.Q OR F_trig_3klik.Q, PT := t#10s);
Q_vypnuti_ukonceno := T_vypnuti_ukonceno.Q;
(* Network 66 *)
TON_blok_OUT16(IN := blok_OUT16, PT := t#500ms);
IF TON_blok_OUT16.Q THEN blok_OUT16 := FALSE; END_IF;
END_FUNCTION_BLOCK

(* POU Zhasni, ST *)
FUNCTION_BLOCK Zhasni
VAR_INPUT
	wIn: WORD;
	xPresun: BOOL;
END_VAR
VAR_OUTPUT
	xonOUT1: BOOL;
	xonOUT2: BOOL;
	xonOUT3: BOOL;

	xoffOUT1: BOOL;
	xoffOUT2: BOOL;
	xoffOUT3: BOOL;
	wLast: WORD;
	xPresunuto: BOOL;
END_VAR
VAR
	start: BOOL;
	TP1: TP;
	stav: WORD;
	last: WORD;
	F_TRIG5: F_TRIG;
END_VAR
IF xPresun=TRUE THEN
	stav:=wIn;
	start:=TRUE;


CASE stav OF
	2: 	xonOUT2:=TRUE;
		last:=2;
	3: 	xonOUT3:=TRUE;
		last:=3;
END_CASE


IF wLast=0 AND stav=1 THEN
xonOUT1:=TRUE;
last:=1;
END_IF

IF NOT( wLast=0) AND stav=1 THEN
	CASE wLast OF
	1: xoffOUT1:=TRUE;
		last:=0;
	2: xoffOUT2:=TRUE;
		last:=0;
	3: xoffOUT3:=TRUE;
		last:=0;
	END_CASE

END_IF
END_IF

TP1(IN:=start , PT:=t#50ms , Q=> , ET=> );
F_TRIG5(CLK:=TP1.Q , Q=> );
IF F_TRIG5.Q=TRUE THEN
	wLast:=last;
	start:=FALSE;
	xoffOUT1:=FALSE;
	xoffOUT2:=FALSE;
	xoffOUT3:=FALSE;
	xonOUT1:=FALSE;
	xonOUT2:=FALSE;
	xonOUT3:=FALSE;
END_IF

xPresunuto:=xPresun;
END_FUNCTION_BLOCK

(* POU dali/Ovladani_7_8_9, ST *)
FUNCTION_BLOCK Ovladani_7_8_9
VAR_INPUT
	xVstup: BOOL;
	rCidlo: REAL;
	rUroven1: REAL;
	rUroven2: REAL;
	tZpozdeniCidla: TIME;
END_VAR
VAR_OUTPUT
	On_7: BOOL;
	On_8: BOOL;
	On_9: BOOL;
	Off_7: BOOL;
	Off_8: BOOL;
	Off_9: BOOL;
END_VAR
VAR
	Stav7: BOOL;
	Stav8: BOOL;
	Stav9: BOOL;
	StavSvetel: BOOL;
	Zmacknuto: BOOL;
	R_TRIG1: R_TRIG;
	F_TRIG1: F_TRIG;
	BLINK1: BLINK;
	Cidlo_zpozdene: REAL;
END_VAR
R_TRIG1(CLK:=xVstup, Q=>Zmacknuto );
F_TRIG1(CLK:=xVstup);
BLINK1(ENABLE:=TRUE , TIMELOW:=tZpozdeniCidla , TIMEHIGH:=t#1s);

IF BLINK1.OUT THEN Cidlo_zpozdene:=rCidlo;
END_IF

StavSvetel:=Stav7 OR Stav8 OR Stav9;

IF Zmacknuto AND (StavSvetel=FALSE) THEN		(*vse zhasnuto*)
	On_7:=TRUE;
	On_8:=TRUE;
	On_9:=TRUE;
	Stav7:=TRUE;
	Stav8:=TRUE;
	Stav9:=TRUE;
END_IF

IF Zmacknuto AND (StavSvetel=TRUE) THEN		(*neco rozsviceno*)
	Off_7:=TRUE;
	Off_8:=TRUE;
	Off_9:=TRUE;
	Stav7:=FALSE;
	Stav8:=FALSE;
	Stav9:=FALSE;
END_IF

IF F_TRIG1.Q THEN
	On_7:=FALSE;
	On_8:=FALSE;
	On_9:=FALSE;
	Off_7:=FALSE;
	Off_8:=FALSE;
	Off_9:=FALSE;
END_IF

IF Cidlo_zpozdene>rUroven1 THEN
	On_7:=FALSE;
	Off_7:=TRUE;
	Stav7:=FALSE;
ELSIF StavSvetel THEN
	On_7:=TRUE;
	Off_7:=FALSE;
	Stav7:=TRUE;
END_IF

IF Cidlo_zpozdene>rUroven2 THEN
	On_9:=FALSE;
	Off_9:=TRUE;
	Stav9:=FALSE;
ELSIF StavSvetel THEN
	On_9:=TRUE;
	Off_9:=FALSE;
	Stav9:=TRUE;
END_IF

IF Zmacknuto AND (StavSvetel=TRUE) THEN		(*neco rozsviceno*)
	Off_7:=TRUE;
	Off_8:=TRUE;
	Off_9:=TRUE;
	Stav7:=FALSE;
	Stav8:=FALSE;
	Stav9:=FALSE;
END_IF

IF F_TRIG1.Q THEN
	On_7:=FALSE;
	On_8:=FALSE;
	On_9:=FALSE;
	Off_7:=FALSE;
	Off_8:=FALSE;
	Off_9:=FALSE;
END_IF
END_FUNCTION_BLOCK

(* POU TriFaze, ST *)
PROGRAM TriFaze
VAR

	Fb750_493_Master3Phase1: Fb750_493_Master3Phase;
	abIn AT %IB22: ARRAY [0..11] OF BYTE;
	abOut AT %QB6: ARRAY [0..11] OF BYTE;

	typ3faze: typConfig3Phase;
	awProud: ARRAY [1..3] OF WORD;
	awNapeti: ARRAY [1..3] OF WORD;
	aiCosFi: ARRAY [1..3] OF INT;
	aiVykon: ARRAY [1..3] OF INT;
	adwSpotreba: ARRAY [1..3] OF DWORD;

	arProud: ARRAY [1..3] OF REAL;
	arNapeti: ARRAY [1..3] OF REAL;
	arCosFi: ARRAY [1..3] OF REAL;
	arVykon: ARRAY [1..3] OF REAL;
	arSpotreba: ARRAY [1..3] OF REAL;
	SmazL1: BOOL;
	SmazL2: BOOL;
	SmazL3: BOOL;
END_VAR
Fb750_493_Master3Phase1(
	xEnable:= TRUE,
	tCycleTime:= ,
	x750_493_000_001:=FALSE ,
	xSaveEnergyConsumption:= ,
	xDeleteEnergyConsumptionL1:=SmazL1 ,
	xDeleteEnergyConsumptionL2:=SmazL1 ,
	xDeleteEnergyConsumptionL3:=SmazL1 ,
	abIn_Data_750_493:=abIn ,
	abOut_Data_750_493:=abOut ,
	typConfig3Phase:=typ3faze ,
	xReady=> ,
	abError=> , 
	awCurrent=>awProud ,
	awVoltage=>awNapeti ,
	aiPowerFactor=>aiCosFi ,
	aiEffectivePower=>aiVykon ,
	adwEnergyConsumption=>adwSpotreba ,
	awMaxCurrent=> , 
	awMaxVoltage=> , 
	awMinCurrent=> ,
	awMinVoltage=> );

arProud[1]:=awProud[1]/1000.0;
arProud[2]:=awProud[2]/1000.0;
arProud[3]:=awProud[3]/1000.0;

arNapeti[1]:=awNapeti[1]/10.0;
arNapeti[2]:=awNapeti[2]/10.0;
arNapeti[3]:=awNapeti[3]/10.0;

arCosFi[1]:=aiCosFi[1]/100.0;
arCosFi[2]:=aiCosFi[2]/100.0;
arCosFi[3]:=aiCosFi[3]/100.0;

arVykon[1]:=aiVykon[1]/10000.0;
arVykon[2]:=aiVykon[2]/10000.0;
arVykon[3]:=aiVykon[3]/10000.0;
;
END_PROGRAM

(* Visualisation Addressing
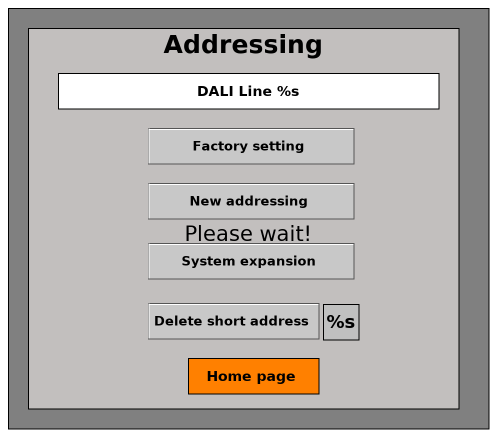
rectangle at (185,80)-(616,461): text "Addressing"
button at (305,235)-(511,271): text "New addressing"; taps DALI_Config.NewAddress; tooltip You have to click and hold the button "New Addressing" longer than two seconds to start the new addressing.
button at (305,295)-(511,331): text "System expansion"; taps DALI_Config.xErweitert; tooltip If you click the button "System expansion", only the ECGs with no short address will be addressed.
rectangle at (480,356)-(516,392): text "%s"; shows DALI_Config.LoeschKurzadr; tooltip Enter the short address to be deleted (1 - 64).; editable
rounded rectangle at (345,410)-(476,446): text "Home page"; opens DALI; tooltip Back to home page
button at (305,180)-(511,216): text "Factory setting"; taps DALI_Config.Reset; tooltip To reset the ECG you have to click and hold the button two seconds. Group and scene configurations will be deleted.
button at (305,355)-(476,391): text "Delete short address"; taps DALI_Config.Loeschen; tooltip The selected short address will be deleted.
rectangle at (265,100)-(546,471): text "Please wait!"; invisible if not DALI_Config.JobMerker[5]
rounded rectangle at (215,125)-(596,161): text "DALI Line %s"; shows DALI_Config.bDali_Linie; tooltip You can change the DALI Line only on the home page.
1 more shapes without text or variables
*)

(* Visualisation DALI
